(* PLC project poST.project, poSTIDE *)
(* stored: creationDateTime 2021-08-31T00:00:00.000000 *)

FUNCTION MOD : ANY_NUM
  VAR_INPUT
    in1 : ANY_INT;
    in2 : ANY_INT;
  END_VAR

END_FUNCTION
